{attribute 'qualified_only'}
{attribute 'strict'}
TYPE eTcoEvaluateMeasurementTestList : (
    None := 0,
    Init := 10,
    Evaluate := 20
);
END_TYPE

(* stored: Version 1.1.0.1, ProductVersion 3.1.4024.10
   DUT eTcoEvaluateMeasurementTestList: Id {c374f53a-e5f0-01ae-3015-c7586dedc47c} *)
